// TIA Portal V20 export
// export: Created 2025-12-01T14:57:44.7272966Z, ExportSetting None, DisplayName Totally Integrated Automation Portal, DisplayVersion V20 Update 3, DisplayName TIA Portal Openness, DisplayVersion V20 Update 3, DisplayName TIA Portal Version Control Interface, DisplayVersion V20 Update 3, DisplayName STEP 7 Professional, DisplayVersion V20 Update 3, DisplayName STEP 7 Safety, DisplayVersion V20 Update 2, DisplayName WinCC Basic/Comfort/Advanced, DisplayVersion V20 Update 3, DisplayName WinCC Professional, DisplayVersion V20 Update 3, DisplayName WinCC Unified, DisplayVersion V20 Update 3
FUNCTION "FC715_Router_BuscarEtiqueta_Lint" : Void   // FC715, SCL
{ S7_Optimized_Access := 'TRUE' }
// stored: AutoNumber false, SetENOAutomatically false
   VAR_INPUT
      Etiqueta : ULInt;   // Etiqueta A Buscar en la Base de Datos
   END_VAR
   VAR_OUTPUT
      Posicion_BBDD : UInt;   // Posición de la Etiqueta (UT) en la Base de Datos. la pos -1 significa que no hay hueco
   END_VAR
   VAR_TEMP
      Cola : UDInt;
      EtiquetaTMP : ULInt;
      Posicion_Etiqueta_TMP : UInt;
      aux_pos : UInt;
   END_VAR
BEGIN
   REGION inicilizar

       #EtiquetaTMP := #Etiqueta;
       #Posicion_Etiqueta_TMP := 0;

   END_REGION
   REGION comprobar_etiqueta

       IF #EtiquetaTMP = 0 THEN
           #Posicion_BBDD := 0;
           RETURN;
       ELSE
           IF #EtiquetaTMP = -1 THEN
               #Posicion_BBDD := -1;
               GOTO busca_pos_libre;
           ELSE

               #Cola := #EtiquetaTMP MOD "ROUT_N_Colas";
               // calculamos el numero de cola
           END_IF;
       END_IF;
   END_REGION

   #Posicion_Etiqueta_TMP := "DB212_Cola_Activa".Cola[#Cola];

   // comprobamos si existe alguna etiqueta en esa cola

   elegir_db_busqueda:
   IF #Posicion_Etiqueta_TMP = 0 THEN
       #Posicion_BBDD := 0;
       RETURN;
   END_IF;


   REGION elegir_db_busqueda
       CASE #Posicion_Etiqueta_TMP OF
           1..1000:
               GOTO busca_1_999;
           1001..2000:
               GOTO busca_1k;
           2001..3000:
               GOTO busca_2k;
           3001..4000:
               GOTO busca_3k;
           ELSE
               #Posicion_BBDD := 0;
               RETURN;
       END_CASE;
   END_REGION

   ////////////////////////////////////////////
   REGION busca_1_a_1000
   busca_1_999:
       IF #EtiquetaTMP = "DB201_RegEtiquetas_0001_1000".Reg_Etiqueta[#Posicion_Etiqueta_TMP].CDB THEN
           #Posicion_BBDD := #Posicion_Etiqueta_TMP;
           RETURN;
       ELSE
           #Posicion_Etiqueta_TMP := "DB201_RegEtiquetas_0001_1000".Reg_Etiqueta[#Posicion_Etiqueta_TMP].Posterior;
           GOTO elegir_db_busqueda;
       END_IF;
   END_REGION

   ////////////////////////////////////////////
   REGION busca_1001_a_2000
   busca_1k:
       #Posicion_Etiqueta_TMP := #Posicion_Etiqueta_TMP - 1000;
       IF #EtiquetaTMP = "DB202_RegEtiquetas_1001_2000".Reg_Etiqueta[#Posicion_Etiqueta_TMP].CDB THEN
           #Posicion_BBDD := #Posicion_Etiqueta_TMP + 1000;
           RETURN;
       ELSE
           #Posicion_Etiqueta_TMP := "DB202_RegEtiquetas_1001_2000".Reg_Etiqueta[#Posicion_Etiqueta_TMP].Posterior;
           GOTO elegir_db_busqueda;
       END_IF;
   END_REGION

   ////////////////////////////////////////////
   REGION busca_2001_a_3000
   busca_2k:
       #Posicion_Etiqueta_TMP := #Posicion_Etiqueta_TMP - 2000;
       IF #EtiquetaTMP = "DB203_RegEtiquetas_2001_3000".Reg_Etiqueta[#Posicion_Etiqueta_TMP].CDB THEN
           #Posicion_BBDD := #Posicion_Etiqueta_TMP + 2000;
           RETURN;
       ELSE
           #Posicion_Etiqueta_TMP := "DB203_RegEtiquetas_2001_3000".Reg_Etiqueta[#Posicion_Etiqueta_TMP].Posterior;
           GOTO elegir_db_busqueda;
       END_IF;

   END_REGION

   ////////////////////////////////////////////
   REGION busca_3001_a_4000
   busca_3k:
       #Posicion_Etiqueta_TMP := #Posicion_Etiqueta_TMP - 3000;
       IF #EtiquetaTMP = "DB204_RegEtiquetas_3001_4000".Reg_Etiqueta[#Posicion_Etiqueta_TMP].CDB THEN
           #Posicion_BBDD := #Posicion_Etiqueta_TMP + 3000;
           RETURN;
       ELSE
           #Posicion_Etiqueta_TMP := "DB204_RegEtiquetas_3001_4000".Reg_Etiqueta[#Posicion_Etiqueta_TMP].Posterior;
           GOTO elegir_db_busqueda;
       END_IF
       ;
   END_REGION
   REGION BUSCA_POS_LIBRE
       // SI LA ETIQUETA DE BUSQUEDA ES -1, VAMOS A SUPONER QUE ESTAMOS BUSCANDO LA PRIMERA POSICION LIBRE EN LA BBDD
   busca_pos_libre:
   FOR #aux_pos := 1 TO 1000 DO
       IF "DB201_RegEtiquetas_0001_1000".Reg_Etiqueta[#aux_pos].CDB = 0 THEN
           #Posicion_BBDD := #aux_pos;
           RETURN;
       END_IF;
   END_FOR;

   FOR #aux_pos := 1 TO 1000 DO
       IF "DB202_RegEtiquetas_1001_2000".Reg_Etiqueta[#aux_pos].CDB = 0 THEN
           #Posicion_BBDD := #aux_pos + 1000;
           RETURN;
       END_IF;
   END_FOR;
   FOR #aux_pos := 1 TO 1000 DO
       IF "DB203_RegEtiquetas_2001_3000".Reg_Etiqueta[#aux_pos].CDB = 0 THEN
           #Posicion_BBDD := #aux_pos + 2000;
           RETURN;
       END_IF;
   END_FOR;
   FOR #aux_pos := 1 TO 1000 DO
       IF "DB204_RegEtiquetas_3001_4000".Reg_Etiqueta[#aux_pos].CDB = 0 THEN
           #Posicion_BBDD := #aux_pos + 3000;
           RETURN;
       END_IF;
   END_FOR;

   END_REGION
END_FUNCTION
